FUNCTION_BLOCK A2X_TO_A2X2 (* Composite FB for convert unidirectional A2X to bidirectional A2X2 *)
  (* Standard: 61499-2; Function: A2X_IN publishes UP/DOWN onto the outgoing (EO_UP/EO_DOWN) side of A2X2_BIDIR. Whatever A2X2_BIDIR receives on its incoming (EI_UP/EI_DOWN) side is forwarded out again as a plain unidirectional signal via A2X_OUT.; Description: Copyright (c) 2026 HR Agrartechnik GmbH This program and the accompanying materials are made available under the terms of the Eclipse Public License 2.0 which is available at https://www.eclipse.org/legal/epl-2.0/ SPDX-License-Identifier: EPL-2.0 *)
  (* Version 1.0, 2026-08-31, Franz Höpfinger, HR Agrartechnik GmbH, Initial Version *)
  PACKAGE adapter::conversion::bidirectional;
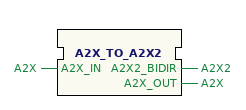
  SOCKETS
    A2X_IN : adapter::types::unidirectional::A2X; (* Adapter Input: unidirectional UP/DOWN source *)
  END_SOCKETS
  PLUGS
    A2X2_BIDIR : adapter::types::bidirectional::A2X2; (* Adapter Output: bidirectional tap, outgoing side driven by A2X_IN, incoming side forwarded to A2X_OUT *)
    A2X_OUT : adapter::types::unidirectional::A2X; (* Adapter Output: mirrors A2X2_BIDIR's incoming (request) side *)
  END_PLUGS
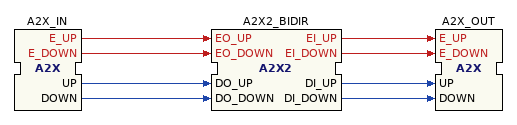
  EVENT_CONNECTIONS
    A2X_IN.E_UP TO A2X2_BIDIR.EO_UP;
    A2X_IN.E_DOWN TO A2X2_BIDIR.EO_DOWN;
    A2X2_BIDIR.EI_UP TO A2X_OUT.E_UP;
    A2X2_BIDIR.EI_DOWN TO A2X_OUT.E_DOWN;
  END_CONNECTIONS
  DATA_CONNECTIONS
    A2X_IN.UP TO A2X2_BIDIR.DO_UP;
    A2X_IN.DOWN TO A2X2_BIDIR.DO_DOWN;
    A2X2_BIDIR.DI_UP TO A2X_OUT.UP;
    A2X2_BIDIR.DI_DOWN TO A2X_OUT.DOWN;
  END_CONNECTIONS
END_FUNCTION_BLOCK
